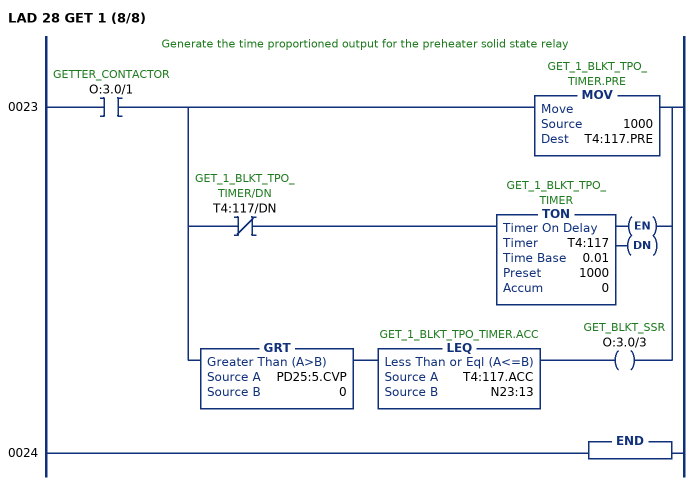
% Rung: 23 %
% Generate the time proportioned output for the preheater solid state relay %
SOR XIC O:3.0/1 BST MOV 1000 T4:117.PRE NXB XIO T4:117/DN TON T4:117 0.01 1000 0 NXB GRT PD25:5.CVP 0 LEQ T4:117.ACC N23:13 OTE O:3.0/3 BND EOR
%   O:3.0/1  GETTER_CONTACTOR %
%   T4:117  GET_1_BLKT_TPO_TIMER %
%   N23:13  GET_1_BLKT_OUTPUT %
%   O:3.0/3  GET_BLKT_SSR %
% Rung: 24 %
SOR END EOR

LADDER 29 "P CONVERT"    % Pressure Unit Conversions %
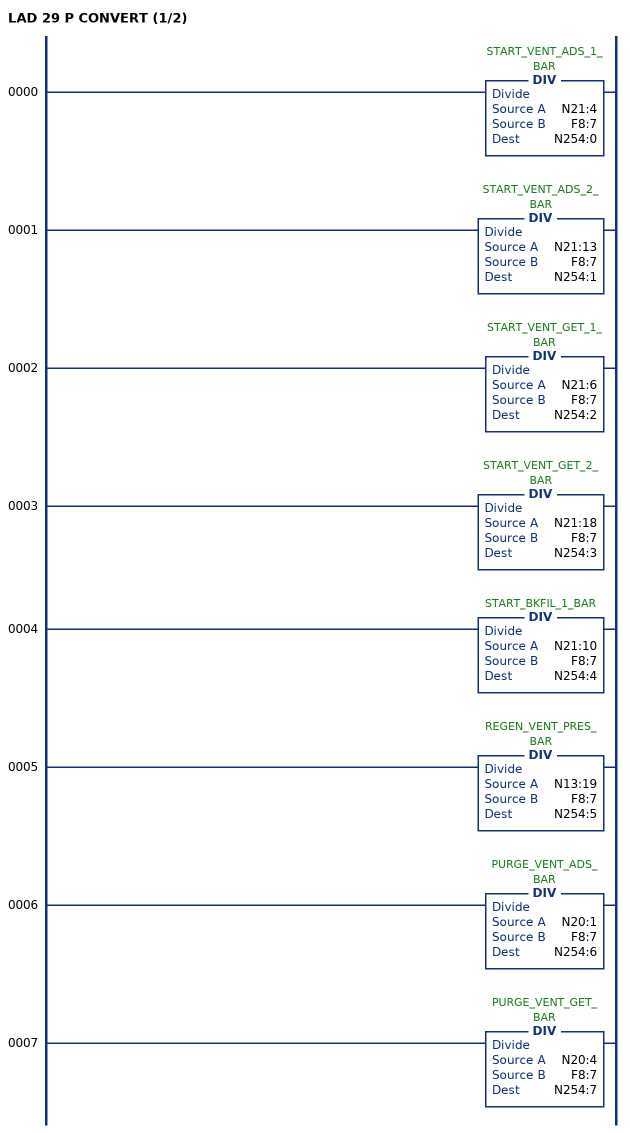
% Rung: 0 %
SOR DIV N21:4 F8:7 N254:0 EOR
%   N21:4  START_VENT_ADS_1_PRS %
%   F8:7  BAR_DIV_FLOAT %
%   N254:0  START_VENT_ADS_1_BAR %
% Rung: 1 %
SOR DIV N21:13 F8:7 N254:1 EOR
%   N21:13  START_VENT_ADS_2_PRS %
%   F8:7  BAR_DIV_FLOAT %
%   N254:1  START_VENT_ADS_2_BAR %
% Rung: 2 %
SOR DIV N21:6 F8:7 N254:2 EOR
%   N21:6  START_VENT_GET_1_PRS %
%   F8:7  BAR_DIV_FLOAT %
%   N254:2  START_VENT_GET_1_BAR %
% Rung: 3 %
SOR DIV N21:18 F8:7 N254:3 EOR
%   N21:18  START_VENT_GET_2_PRS %
%   F8:7  BAR_DIV_FLOAT %
%   N254:3  START_VENT_GET_2_BAR %
% Rung: 4 %
SOR DIV N21:10 F8:7 N254:4 EOR
%   N21:10  START_BKFIL_1_PRS %
%   F8:7  BAR_DIV_FLOAT %
%   N254:4  START_BKFIL_1_BAR %
% Rung: 5 %
SOR DIV N13:19 F8:7 N254:5 EOR
%   N13:19  REGEN_VENT_PRES %
%   F8:7  BAR_DIV_FLOAT %
%   N254:5  REGEN_VENT_PRES_BAR %
% Rung: 6 %
SOR DIV N20:1 F8:7 N254:6 EOR
%   N20:1  PURGE_VENT_ADS_PRES %
%   F8:7  BAR_DIV_FLOAT %
%   N254:6  PURGE_VENT_ADS_BAR %
% Rung: 7 %
SOR DIV N20:4 F8:7 N254:7 EOR
%   N20:4  PURGE_VENT_GET_PRES %
%   F8:7  BAR_DIV_FLOAT %
%   N254:7  PURGE_VENT_GET_BAR %

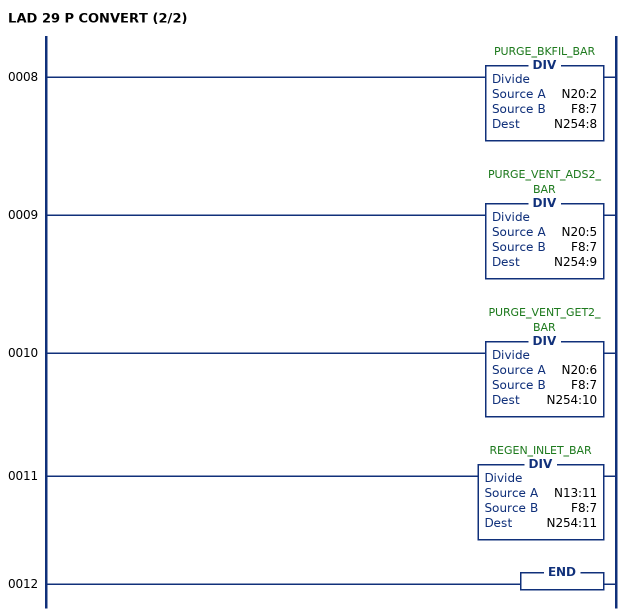
% Rung: 8 %
SOR DIV N20:2 F8:7 N254:8 EOR
%   N20:2  PURGE_BKFIL_PRES %
%   F8:7  BAR_DIV_FLOAT %
%   N254:8  PURGE_BKFIL_BAR %
% Rung: 9 %
SOR DIV N20:5 F8:7 N254:9 EOR
%   N20:5  PURGE_VENT_ADS_2_PX %
%   F8:7  BAR_DIV_FLOAT %
%   N254:9  PURGE_VENT_ADS2_BAR %
% Rung: 10 %
SOR DIV N20:6 F8:7 N254:10 EOR
%   N20:6  PURGE_VENT_GET_2_PX %
%   F8:7  BAR_DIV_FLOAT %
%   N254:10  PURGE_VENT_GET2_BAR %
% Rung: 11 %
SOR DIV N13:11 F8:7 N254:11 EOR
%   N13:11  REGEN_INLET_PSIG %
%   F8:7  BAR_DIV_FLOAT %
%   N254:11  REGEN_INLET_BAR %
% Rung: 12 %
SOR END EOR

LADDER 49 "MODBUS"
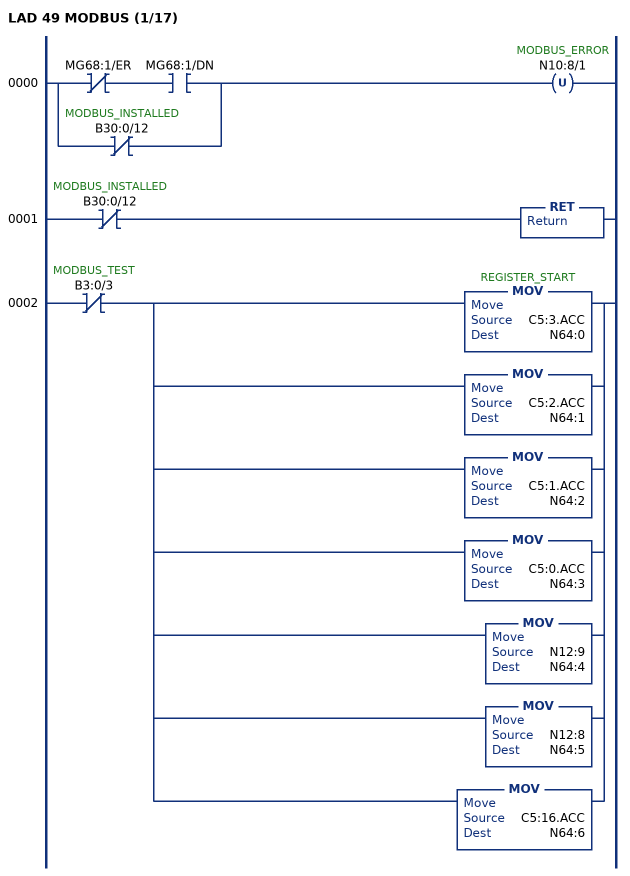
% Rung: 0 %
SOR BST XIO MG68:1/ER XIC MG68:1/DN NXB XIO B30:0/12 BND OTU N10:8/1 EOR
%   B30:0/12  MODBUS_INSTALLED %
%   N10:8/1  MODBUS_ERROR %
% Rung: 1 %
SOR XIO B30:0/12 RET EOR
%   B30:0/12  MODBUS_INSTALLED %
% Rung: 2 %
SOR XIO B3:0/3 BST MOV C5:3.ACC N64:0 NXB MOV C5:2.ACC N64:1 NXB MOV C5:1.ACC N64:2 NXB MOV C5:0.ACC N64:3 NXB MOV N12:9 N64:4 NXB MOV N12:8 N64:5 NXB MOV C5:16.ACC N64:6 BND EOR
%   B3:0/3  MODBUS_TEST %
%   C5:3  PURIFY_ACTIVE_TTL_DY  "COUNTER The number of total elapsed purification days for the process equipment" %
%   N64:0  REGISTER_START %
%   C5:2  PURIFY_ACTIVE_TTL_HR  "COUNTER The number of total elapsed purification hours for the process equipment" %
%   C5:1  PURIFY_ACTIVE_MINUTE  "COUNTER The number of elapsed purification minutes for the current ADS (60 min)" %
%   C5:0  PURIFY_ACTIVE_HOURS  "COUNTER The number of elapsed purification hours for the current ADS" %
%   N12:9  MIN_LEFT_IN_PURIFY %
%   N12:8  HRS_LEFT_IN_PURIFY %
%   C5:16  GETTER_SERVICE_DAYS %

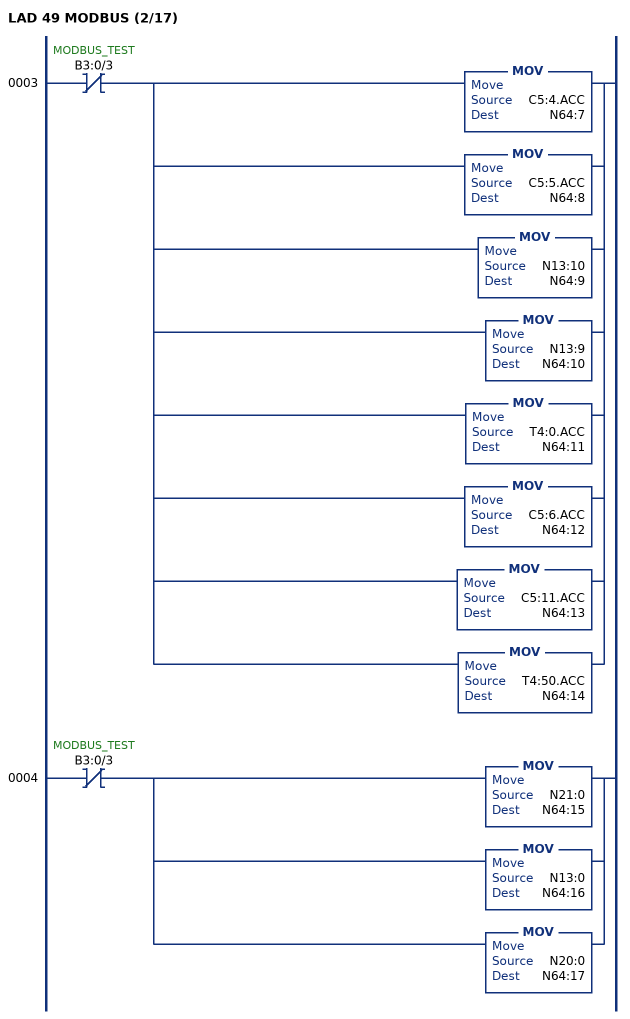
% Rung: 3 %
SOR XIO B3:0/3 BST MOV C5:4.ACC N64:7 NXB MOV C5:5.ACC N64:8 NXB MOV N13:10 N64:9 NXB MOV N13:9 N64:10 NXB MOV T4:0.ACC N64:11 NXB MOV C5:6.ACC N64:12 NXB MOV C5:11.ACC N64:13 NXB MOV T4:50.ACC N64:14 BND EOR
%   B3:0/3  MODBUS_TEST %
%   C5:4  REGEN_RUN_MINUTE %
%   C5:5  REGEN_COOL_MINUTE  "COUNTER Regen the number of minutes for which the bed has cooled" %
%   N13:10  REGEN_MIN_LEFT  "STATUS Preheater Alarm Measured temperature change" %
%   N13:9  REGEN_HRS_LEFT  "STATUS Regen Preheater Temperature Initial Temperature" %
%   T4:0  PURIFY_OVERLAP_TIMER  "TIMER Purify Overlap" %
%   C5:6  START_PURGE_CTR %
%   C5:11  H2_LEAK_RST_MIN %
%   T4:50  H2_LEAK_RST_SEC %
% Rung: 4 %
SOR XIO B3:0/3 BST MOV N21:0 N64:15 NXB MOV N13:0 N64:16 NXB MOV N20:0 N64:17 BND EOR
%   B3:0/3  MODBUS_TEST %
%   N21:0  START_STATE %
%   N13:0  REGEN_STATE  "STATE The current state of the regen process" %
%   N20:0  PURGE_STATE %

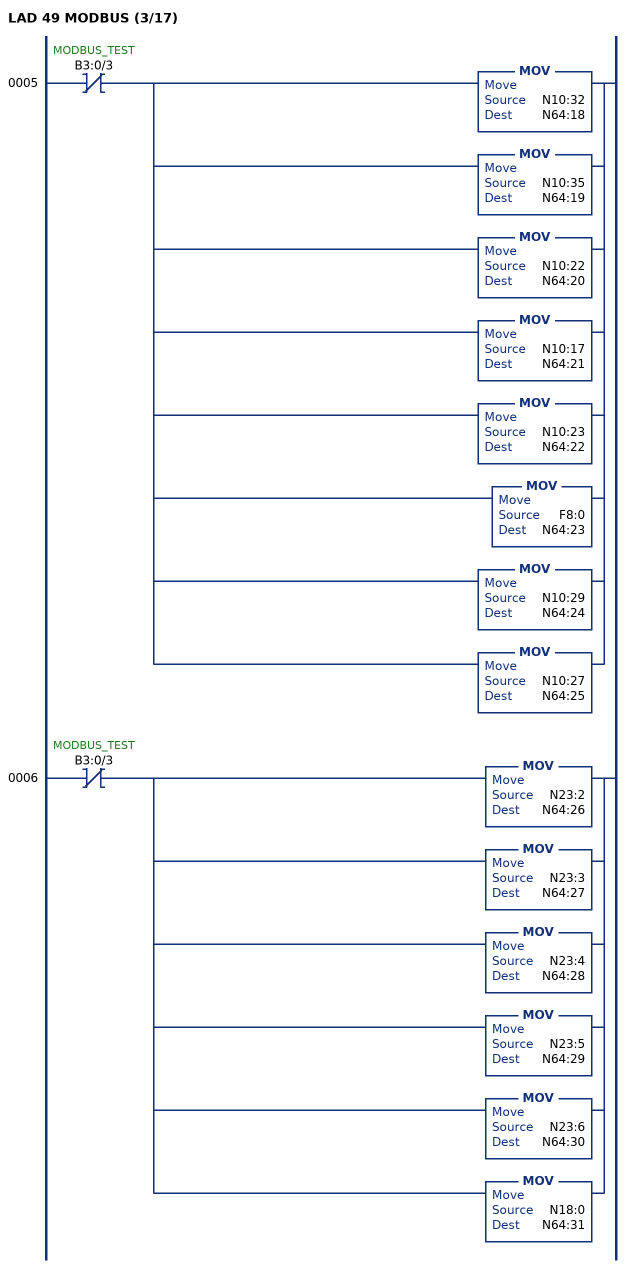
% Rung: 5 %
SOR XIO B3:0/3 BST MOV N10:32 N64:18 NXB MOV N10:35 N64:19 NXB MOV N10:22 N64:20 NXB MOV N10:17 N64:21 NXB MOV N10:23 N64:22 NXB MOV F8:0 N64:23 NXB MOV N10:29 N64:24 NXB MOV N10:27 N64:25 BND EOR
%   B3:0/3  MODBUS_TEST %
%   N10:32  ADS_A_INLET_PX_PRES %
%   N10:35  ADS_B_INLET_PX_PRES %
%   N10:22  OUTLET_PX_PRESSURE %
%   N10:17  INLET_PX_PRESSURE %
%   N10:23  H2_LEVEL_PERCENT %
%   F8:0  MFM_CUM_HR %
%   N10:29  MFC_SLPM %
%   N10:27  MFC_SETPOINT %
% Rung: 6 %
SOR XIO B3:0/3 BST MOV N23:2 N64:26 NXB MOV N23:3 N64:27 NXB MOV N23:4 N64:28 NXB MOV N23:5 N64:29 NXB MOV N23:6 N64:30 NXB MOV N18:0 N64:31 BND EOR
%   B3:0/3  MODBUS_TEST %
%   N23:2  GET_1_PH_INNER_TEMP %
%   N23:3  GET_1_PH_OUTER_TEMP %
%   N23:4  GET_1_PH_GAS_TEMP %
%   N23:5  GET_1_VSL_WALL_TEMP %
%   N23:6  GET_1_VSL_BED_TEMP %
%   N18:0  GET_VSL_OUT_GAS_TEMP %

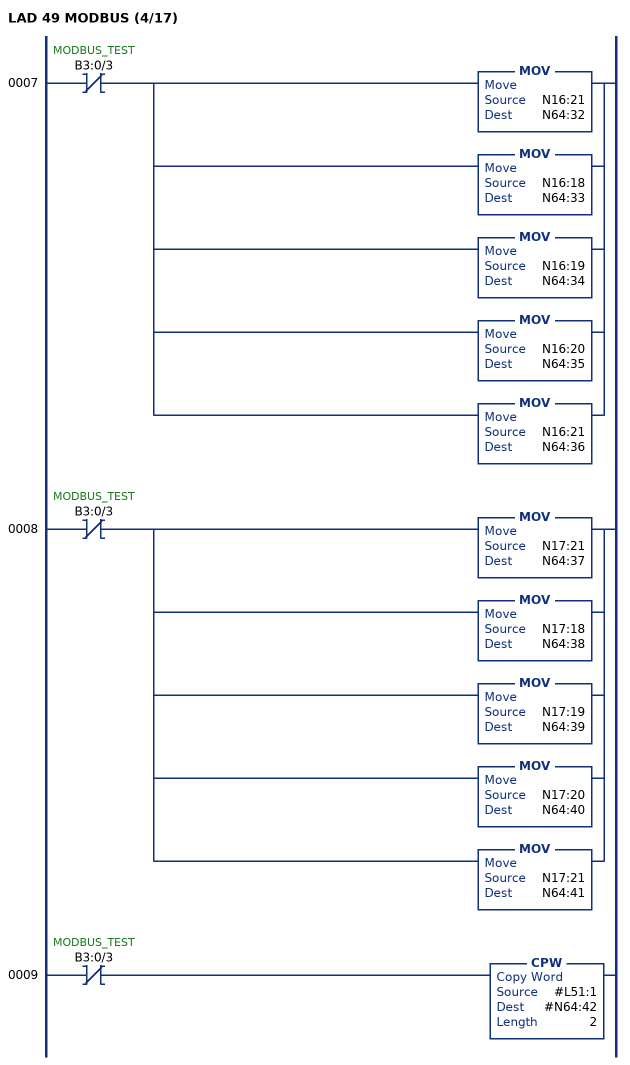
% Rung: 7 %
SOR XIO B3:0/3 BST MOV N16:21 N64:32 NXB MOV N16:18 N64:33 NXB MOV N16:19 N64:34 NXB MOV N16:20 N64:35 NXB MOV N16:21 N64:36 BND EOR
%   B3:0/3  MODBUS_TEST %
%   N16:21  ADS_A_BED_TEMP_READ %
%   N16:18  PH_A_WALL_TEMP_READ %
%   N16:19  PH_A_GAS_TEMP_READ %
%   N16:20  ADS_A_WALL_TEMP_READ %
% Rung: 8 %
SOR XIO B3:0/3 BST MOV N17:21 N64:37 NXB MOV N17:18 N64:38 NXB MOV N17:19 N64:39 NXB MOV N17:20 N64:40 NXB MOV N17:21 N64:41 BND EOR
%   B3:0/3  MODBUS_TEST %
%   N17:21  ADS_B_BED_TEMP_READ %
%   N17:18  PH_B_WALL_TEMP_READ %
%   N17:19  PH_B_GAS_TEMP_READ %
%   N17:20  ADS_B_WALL_TEMP_READ %
% Rung: 9 %
SOR XIO B3:0/3 CPW #L51:1 #N64:42 2 EOR
%   B3:0/3  MODBUS_TEST %
%   L51:1  TOTAL_FLOW_MODBUS %

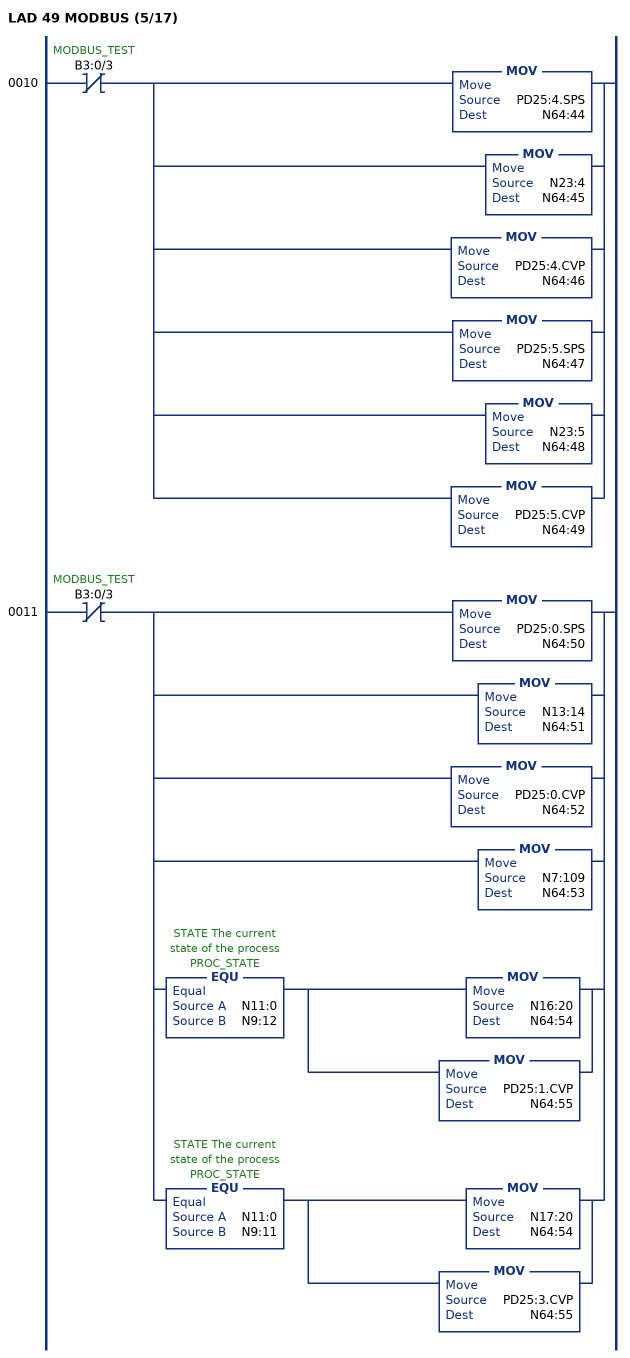
% Rung: 10 %
SOR XIO B3:0/3 BST MOV PD25:4.SPS N64:44 NXB MOV N23:4 N64:45 NXB MOV PD25:4.CVP N64:46 NXB MOV PD25:5.SPS N64:47 NXB MOV N23:5 N64:48 NXB MOV PD25:5.CVP N64:49 BND EOR
%   B3:0/3  MODBUS_TEST %
%   N23:4  GET_1_PH_GAS_TEMP %
%   N23:5  GET_1_VSL_WALL_TEMP %
% Rung: 11 %
SOR XIO B3:0/3 BST MOV PD25:0.SPS N64:50 NXB MOV N13:14 N64:51 NXB MOV PD25:0.CVP N64:52 NXB MOV N7:109 N64:53 NXB EQU N11:0 N9:12 BST MOV N16:20 N64:54 NXB MOV PD25:1.CVP N64:55 BND NXB EQU N11:0 N9:11 BST MOV N17:20 N64:54 NXB MOV PD25:3.CVP N64:55 BND BND EOR
%   B3:0/3  MODBUS_TEST %
%   N13:14  ADS_PH_GAS_TC %
%   N7:109  BLANKET_SP  "CONTROL Blanket PID Setpoint" %
%   N11:0  PROC_STATE  "STATE The current state of the process" %
%   N9:12  PROC_PFY_B_REG_A  "STATE Process Purify B" %
%   N16:20  ADS_A_WALL_TEMP_READ %
%   N9:11  PROC_PFY_A_REG_B  "STATE Process Purify A" %
%   N17:20  ADS_B_WALL_TEMP_READ %

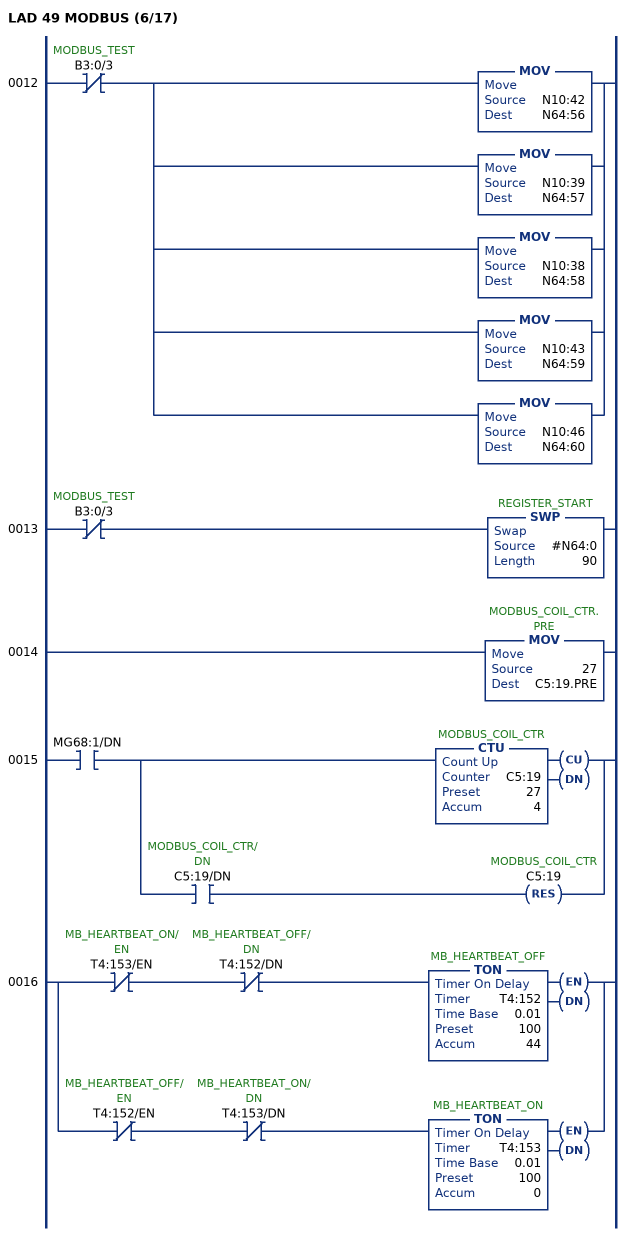
% Rung: 12 %
SOR XIO B3:0/3 BST MOV N10:42 N64:56 NXB MOV N10:39 N64:57 NXB MOV N10:38 N64:58 NXB MOV N10:43 N64:59 NXB MOV N10:46 N64:60 BND EOR
%   B3:0/3  MODBUS_TEST %
%   N10:42  ARGON_PX_PRESS %
%   N10:39  WATER_FLOW_GPM %
%   N10:38  PNEU_PX_PRESS %
%   N10:43  PIPING_BAY_WC %
%   N10:46  ELEC_CAB_WC %
% Rung: 13 %
SOR XIO B3:0/3 SWP #N64:0 90 EOR
%   B3:0/3  MODBUS_TEST %
%   N64:0  REGISTER_START %
% Rung: 14 %
SOR MOV 27 C5:19.PRE EOR
%   C5:19  MODBUS_COIL_CTR %
% Rung: 15 %
SOR XIC MG68:1/DN BST CTU C5:19 27 4 NXB XIC C5:19/DN RES C5:19 BND EOR
%   C5:19  MODBUS_COIL_CTR %
% Rung: 16 %
SOR BST XIO T4:153/EN XIO T4:152/DN TON T4:152 0.01 100 44 NXB XIO T4:152/EN XIO T4:153/DN TON T4:153 0.01 100 0 BND EOR
%   T4:153  MB_HEARTBEAT_ON %
%   T4:152  MB_HEARTBEAT_OFF %

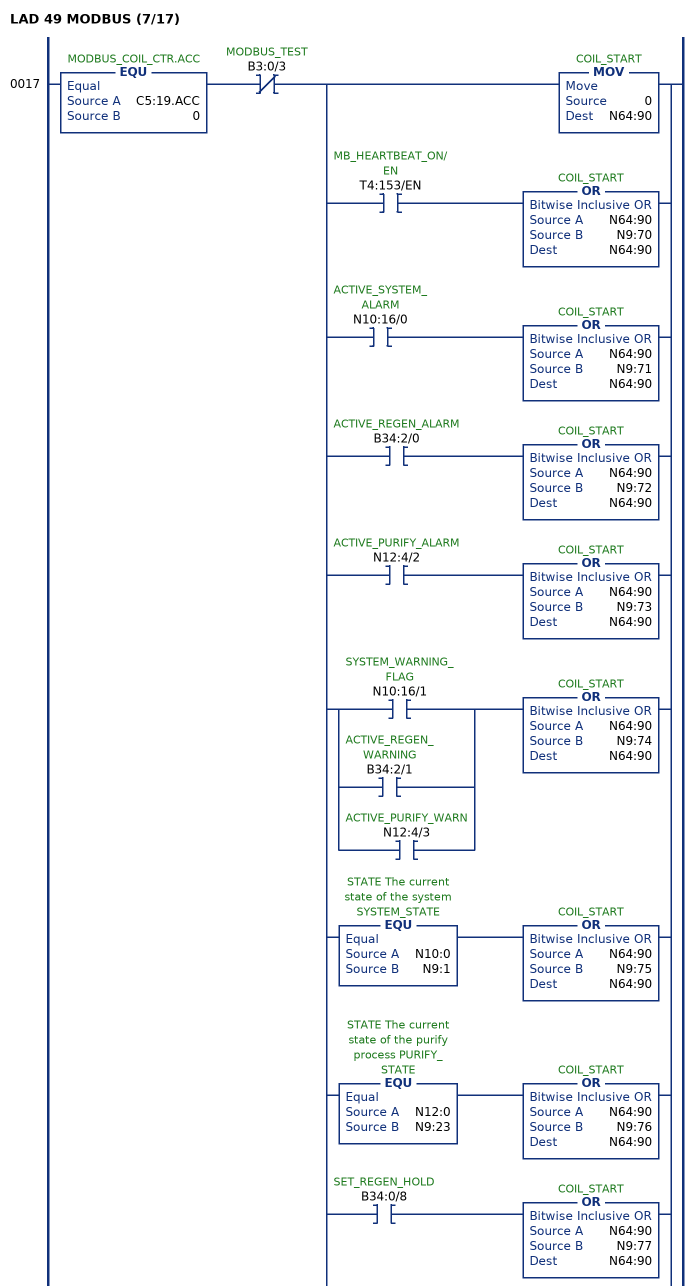

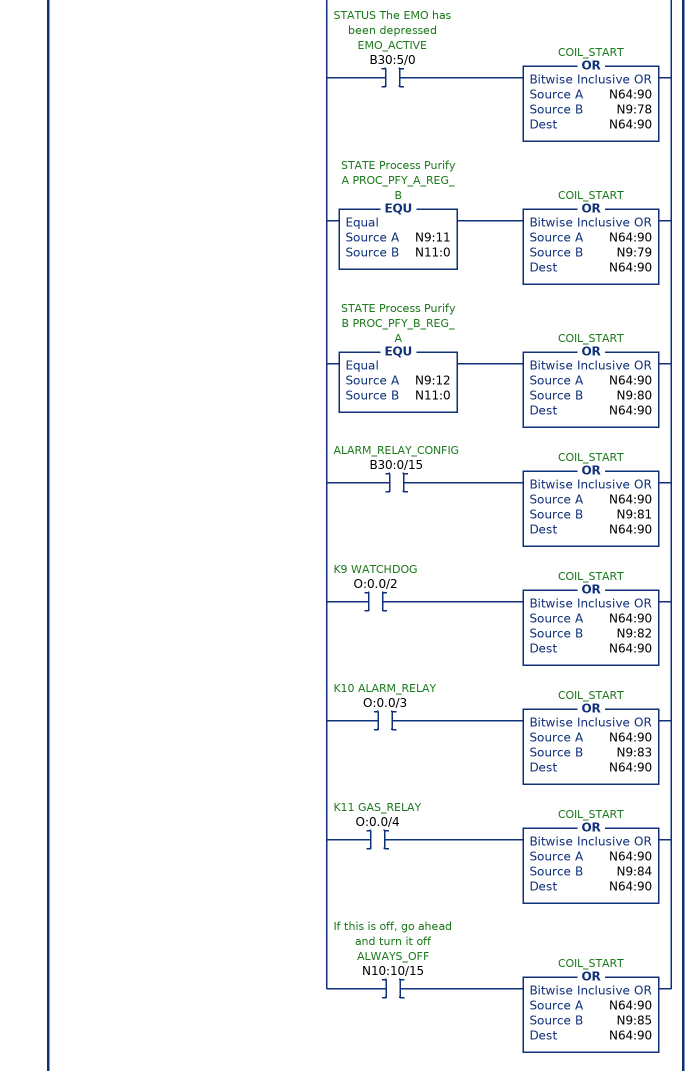
% Rung: 17 %
SOR EQU C5:19.ACC 0 XIO B3:0/3 BST MOV 0 N64:90 NXB XIC T4:153/EN OR N64:90 N9:70 N64:90 NXB XIC N10:16/0 OR N64:90 N9:71 N64:90 NXB XIC B34:2/0 OR N64:90 N9:72 N64:90 NXB XIC N12:4/2 OR N64:90 N9:73 N64:90 NXB BST XIC N10:16/1 NXB XIC B34:2/1 NXB XIC N12:4/3 BND OR N64:90 N9:74 N64:90 NXB EQU N10:0 N9:1 OR N64:90 N9:75 N64:90 NXB EQU N12:0 N9:23 OR N64:90 N9:76 N64:90 NXB XIC B34:0/8 OR N64:90 N9:77 N64:90 NXB XIC B30:5/0 OR N64:90 N9:78 N64:90 NXB EQU N9:11 N11:0 OR N64:90 N9:79 N64:90 NXB EQU N9:12 N11:0 OR N64:90 N9:80 N64:90 NXB XIC B30:0/15 OR N64:90 N9:81 N64:90 NXB XIC O:0.0/2 OR N64:90 N9:82 N64:90 NXB XIC O:0.0/3 OR N64:90 N9:83 N64:90 NXB XIC O:0.0/4 OR N64:90 N9:84 N64:90 NXB XIC N10:10/15 OR N64:90 N9:85 N64:90 BND EOR
%   C5:19  MODBUS_COIL_CTR %
%   B3:0/3  MODBUS_TEST %
%   N64:90  COIL_START %
%   T4:153  MB_HEARTBEAT_ON %
%   N9:70  BIT_0 %
%   N10:16/0  ACTIVE_SYSTEM_ALARM %
%   N9:71  BIT_1 %
%   B34:2/0  ACTIVE_REGEN_ALARM %
%   N9:72  BIT_2 %
%   N12:4/2  ACTIVE_PURIFY_ALARM %
%   N9:73  BIT_3 %
%   N10:16/1  SYSTEM_WARNING_FLAG %
%   B34:2/1  ACTIVE_REGEN_WARNING %
%   N12:4/3  ACTIVE_PURIFY_WARN %
%   N9:74  BIT_4 %
%   N10:0  SYSTEM_STATE  "STATE The current state of the system" %
%   N9:1  SYSTEM_STANDBY  "STATE System Process" %
%   N9:75  BIT_5 %
%   N12:0  PURIFY_STATE  "STATE The current state of the purify process" %
%   N9:23  PURIFY_MANUAL_HOLD  "STATE Purify Manual Hold" %
%   N9:76  BIT_6 %
%   B34:0/8  SET_REGEN_HOLD %
%   N9:77  BIT_7 %
%   B30:5/0  EMO_ACTIVE  "STATUS The EMO has been depressed" %
%   N9:78  BIT_8 %
%   N9:11  PROC_PFY_A_REG_B  "STATE Process Purify A" %
%   N11:0  PROC_STATE  "STATE The current state of the process" %
%   N9:79  BIT_9 %
%   N9:12  PROC_PFY_B_REG_A  "STATE Process Purify B" %
%   N9:80  BIT_10 %
%   B30:0/15  ALARM_RELAY_CONFIG %
%   N9:81  BIT_11 %
%   O:0.0/2  WATCHDOG  "K9" %
%   N9:82  BIT_12 %
%   O:0.0/3  ALARM_RELAY  "K10" %
%   N9:83  BIT_13 %
%   O:0.0/4  GAS_RELAY  "K11" %
%   N9:84  BIT_14 %
%   N10:10/15  ALWAYS_OFF  "If this is off, go ahead and turn it off" %
%   N9:85  BIT_15 %

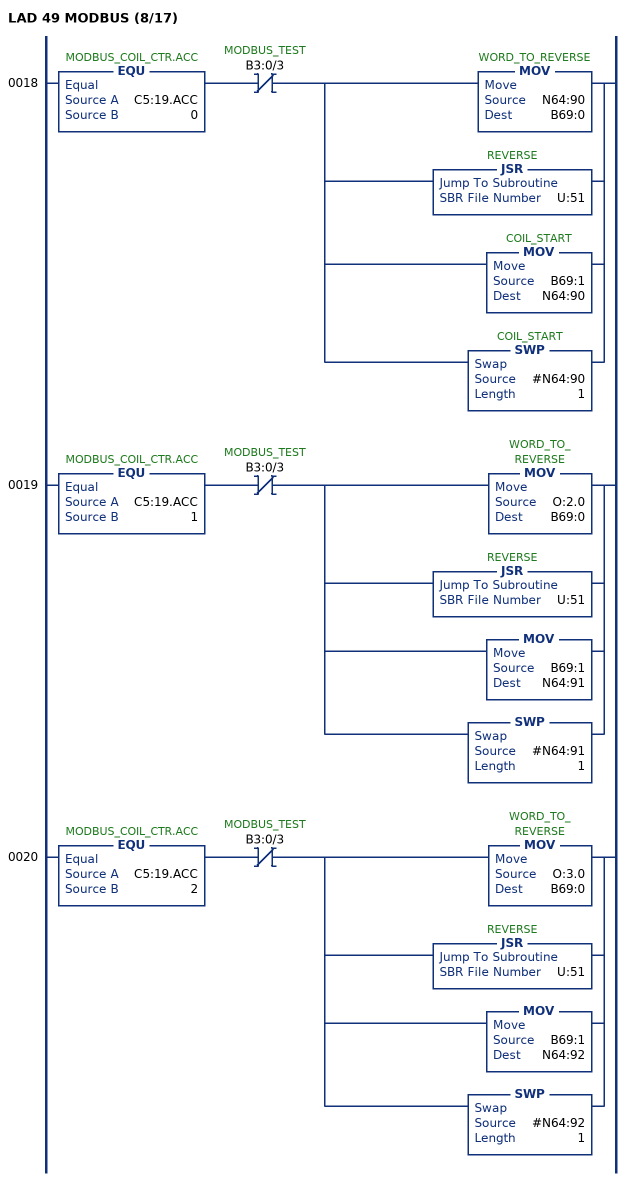
% Rung: 18 %
SOR EQU C5:19.ACC 0 XIO B3:0/3 BST MOV N64:90 B69:0 NXB JSR U:51 NXB MOV B69:1 N64:90 NXB SWP #N64:90 1 BND EOR
%   C5:19  MODBUS_COIL_CTR %
%   B3:0/3  MODBUS_TEST %
%   N64:90  COIL_START %
%   B69:0  WORD_TO_REVERSE %
%   U:51  REVERSE %
%   B69:1  REVERSED_WORD %
% Rung: 19 %
SOR EQU C5:19.ACC 1 XIO B3:0/3 BST MOV O:2.0 B69:0 NXB JSR U:51 NXB MOV B69:1 N64:91 NXB SWP #N64:91 1 BND EOR
%   C5:19  MODBUS_COIL_CTR %
%   B3:0/3  MODBUS_TEST %
%   B69:0  WORD_TO_REVERSE %
%   U:51  REVERSE %
%   B69:1  REVERSED_WORD %
% Rung: 20 %
SOR EQU C5:19.ACC 2 XIO B3:0/3 BST MOV O:3.0 B69:0 NXB JSR U:51 NXB MOV B69:1 N64:92 NXB SWP #N64:92 1 BND EOR
%   C5:19  MODBUS_COIL_CTR %
%   B3:0/3  MODBUS_TEST %
%   B69:0  WORD_TO_REVERSE %
%   U:51  REVERSE %
%   B69:1  REVERSED_WORD %

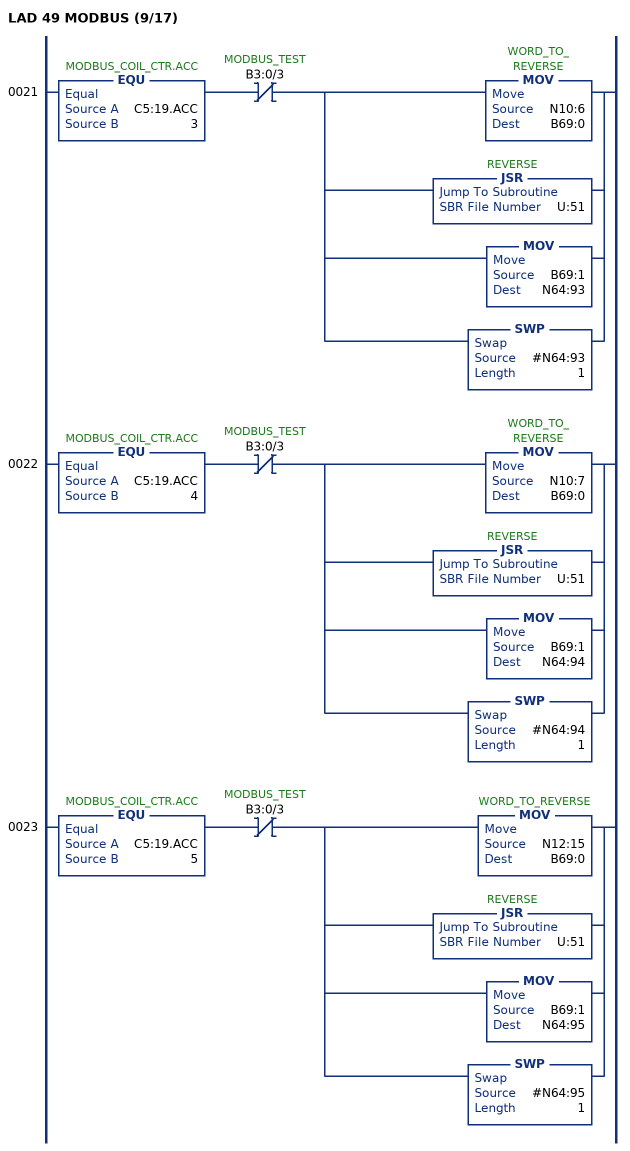
% Rung: 21 %
SOR EQU C5:19.ACC 3 XIO B3:0/3 BST MOV N10:6 B69:0 NXB JSR U:51 NXB MOV B69:1 N64:93 NXB SWP #N64:93 1 BND EOR
%   C5:19  MODBUS_COIL_CTR %
%   B3:0/3  MODBUS_TEST %
%   N10:6  SYSTEM_ALARMS_0  "ALARM System alarms" %
%   B69:0  WORD_TO_REVERSE %
%   U:51  REVERSE %
%   B69:1  REVERSED_WORD %
% Rung: 22 %
SOR EQU C5:19.ACC 4 XIO B3:0/3 BST MOV N10:7 B69:0 NXB JSR U:51 NXB MOV B69:1 N64:94 NXB SWP #N64:94 1 BND EOR
%   C5:19  MODBUS_COIL_CTR %
%   B3:0/3  MODBUS_TEST %
%   N10:7  SYSTEM_ALARMS_1  "ALARM System alarms" %
%   B69:0  WORD_TO_REVERSE %
%   U:51  REVERSE %
%   B69:1  REVERSED_WORD %
% Rung: 23 %
SOR EQU C5:19.ACC 5 XIO B3:0/3 BST MOV N12:15 B69:0 NXB JSR U:51 NXB MOV B69:1 N64:95 NXB SWP #N64:95 1 BND EOR
%   C5:19  MODBUS_COIL_CTR %
%   B3:0/3  MODBUS_TEST %
%   N12:15  PURIFY_ALARMS_0 %
%   B69:0  WORD_TO_REVERSE %
%   U:51  REVERSE %
%   B69:1  REVERSED_WORD %

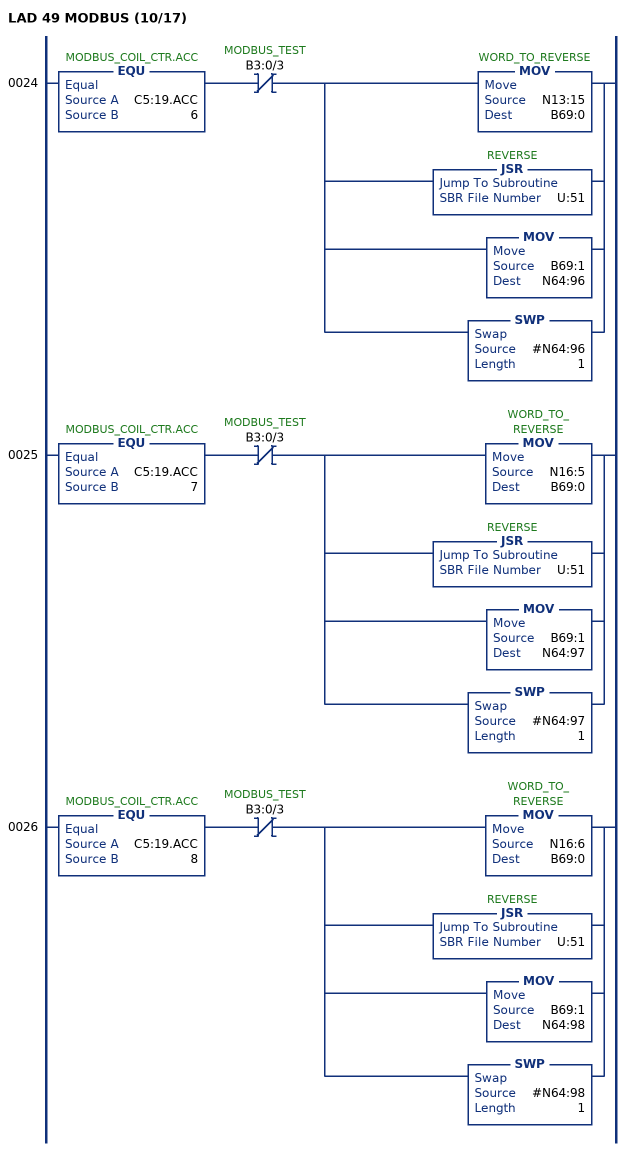
% Rung: 24 %
SOR EQU C5:19.ACC 6 XIO B3:0/3 BST MOV N13:15 B69:0 NXB JSR U:51 NXB MOV B69:1 N64:96 NXB SWP #N64:96 1 BND EOR
%   C5:19  MODBUS_COIL_CTR %
%   B3:0/3  MODBUS_TEST %
%   N13:15  REGEN_ALARMS_0 %
%   B69:0  WORD_TO_REVERSE %
%   U:51  REVERSE %
%   B69:1  REVERSED_WORD %
% Rung: 25 %
SOR EQU C5:19.ACC 7 XIO B3:0/3 BST MOV N16:5 B69:0 NXB JSR U:51 NXB MOV B69:1 N64:97 NXB SWP #N64:97 1 BND EOR
%   C5:19  MODBUS_COIL_CTR %
%   B3:0/3  MODBUS_TEST %
%   N16:5  ADS_A_REGEN_ALARMS_0  "ALARM ADS A Alarms" %
%   B69:0  WORD_TO_REVERSE %
%   U:51  REVERSE %
%   B69:1  REVERSED_WORD %
% Rung: 26 %
SOR EQU C5:19.ACC 8 XIO B3:0/3 BST MOV N16:6 B69:0 NXB JSR U:51 NXB MOV B69:1 N64:98 NXB SWP #N64:98 1 BND EOR
%   C5:19  MODBUS_COIL_CTR %
%   B3:0/3  MODBUS_TEST %
%   N16:6  ADS_A_PURIFY_ALARMS  "ALARM ADS A Alarms" %
%   B69:0  WORD_TO_REVERSE %
%   U:51  REVERSE %
%   B69:1  REVERSED_WORD %

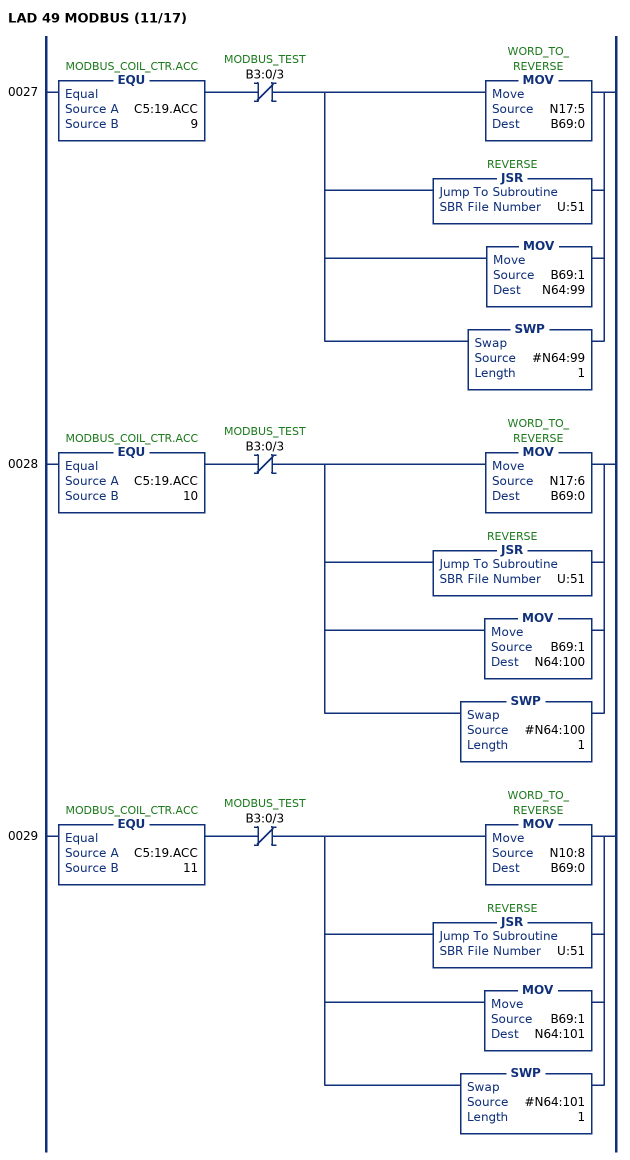
% Rung: 27 %
SOR EQU C5:19.ACC 9 XIO B3:0/3 BST MOV N17:5 B69:0 NXB JSR U:51 NXB MOV B69:1 N64:99 NXB SWP #N64:99 1 BND EOR
%   C5:19  MODBUS_COIL_CTR %
%   B3:0/3  MODBUS_TEST %
%   N17:5  ADS_B_REGEN_ALARMS_0  "ALARM Alarm bits" %
%   B69:0  WORD_TO_REVERSE %
%   U:51  REVERSE %
%   B69:1  REVERSED_WORD %
% Rung: 28 %
SOR EQU C5:19.ACC 10 XIO B3:0/3 BST MOV N17:6 B69:0 NXB JSR U:51 NXB MOV B69:1 N64:100 NXB SWP #N64:100 1 BND EOR
%   C5:19  MODBUS_COIL_CTR %
%   B3:0/3  MODBUS_TEST %
%   N17:6  ADS_B_PURIFY_ALARMS  "ALARM ADS B Alarms" %
%   B69:0  WORD_TO_REVERSE %
%   U:51  REVERSE %
%   B69:1  REVERSED_WORD %
% Rung: 29 %
SOR EQU C5:19.ACC 11 XIO B3:0/3 BST MOV N10:8 B69:0 NXB JSR U:51 NXB MOV B69:1 N64:101 NXB SWP #N64:101 1 BND EOR
%   C5:19  MODBUS_COIL_CTR %
%   B3:0/3  MODBUS_TEST %
%   N10:8  SYSTEM_WARNINGS_0  "WARNING System Warnings" %
%   B69:0  WORD_TO_REVERSE %
%   U:51  REVERSE %
%   B69:1  REVERSED_WORD %

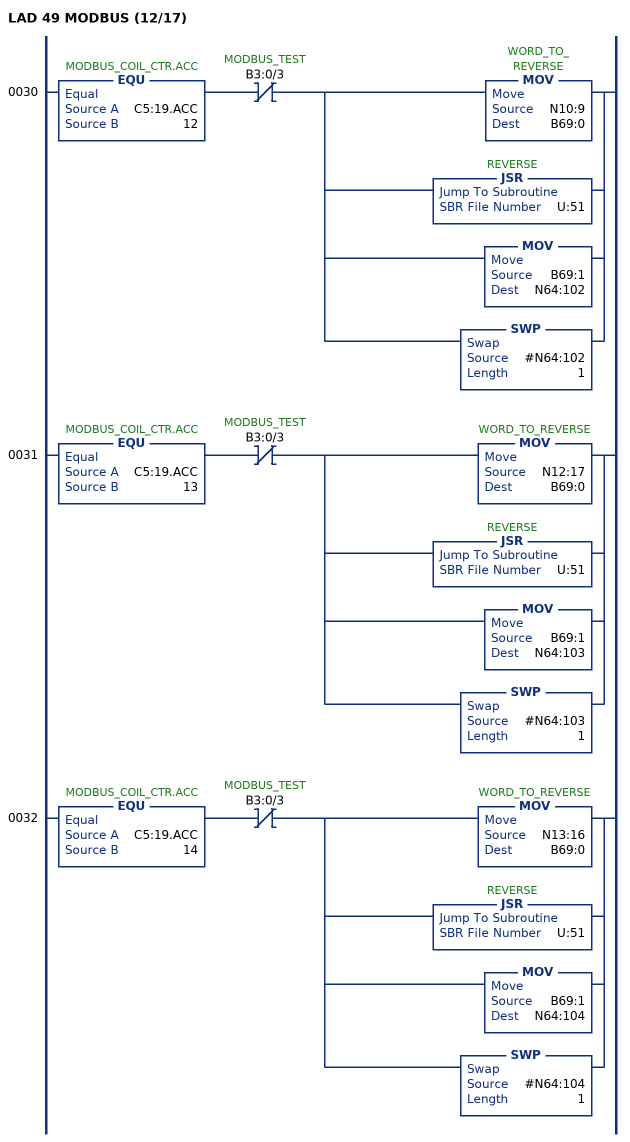
% Rung: 30 %
SOR EQU C5:19.ACC 12 XIO B3:0/3 BST MOV N10:9 B69:0 NXB JSR U:51 NXB MOV B69:1 N64:102 NXB SWP #N64:102 1 BND EOR
%   C5:19  MODBUS_COIL_CTR %
%   B3:0/3  MODBUS_TEST %
%   N10:9  SYSTEM_WARNINGS_1  "WARNING System Warnings" %
%   B69:0  WORD_TO_REVERSE %
%   U:51  REVERSE %
%   B69:1  REVERSED_WORD %
% Rung: 31 %
SOR EQU C5:19.ACC 13 XIO B3:0/3 BST MOV N12:17 B69:0 NXB JSR U:51 NXB MOV B69:1 N64:103 NXB SWP #N64:103 1 BND EOR
%   C5:19  MODBUS_COIL_CTR %
%   B3:0/3  MODBUS_TEST %
%   N12:17  PURIFY_WARNINGS_0 %
%   B69:0  WORD_TO_REVERSE %
%   U:51  REVERSE %
%   B69:1  REVERSED_WORD %
% Rung: 32 %
SOR EQU C5:19.ACC 14 XIO B3:0/3 BST MOV N13:16 B69:0 NXB JSR U:51 NXB MOV B69:1 N64:104 NXB SWP #N64:104 1 BND EOR
%   C5:19  MODBUS_COIL_CTR %
%   B3:0/3  MODBUS_TEST %
%   N13:16  REGEN_WARNINGS_0 %
%   B69:0  WORD_TO_REVERSE %
%   U:51  REVERSE %
%   B69:1  REVERSED_WORD %

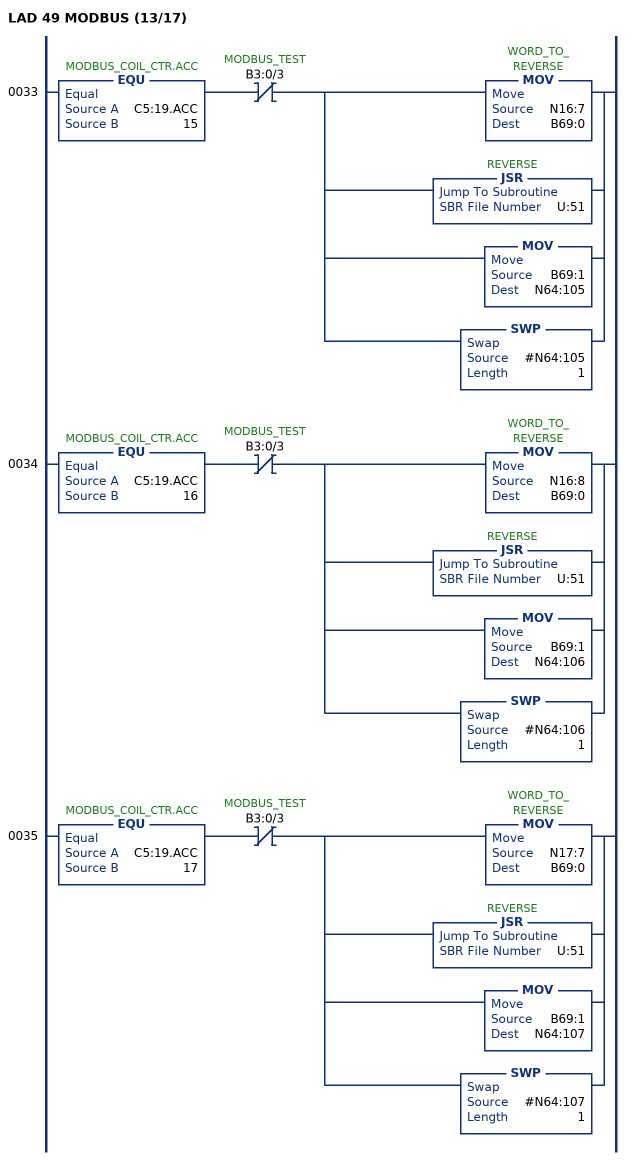
% Rung: 33 %
SOR EQU C5:19.ACC 15 XIO B3:0/3 BST MOV N16:7 B69:0 NXB JSR U:51 NXB MOV B69:1 N64:105 NXB SWP #N64:105 1 BND EOR
%   C5:19  MODBUS_COIL_CTR %
%   B3:0/3  MODBUS_TEST %
%   N16:7  ADS_A_REGEN_WARN_0  "WARNING ADS A Warnings" %
%   B69:0  WORD_TO_REVERSE %
%   U:51  REVERSE %
%   B69:1  REVERSED_WORD %
% Rung: 34 %
SOR EQU C5:19.ACC 16 XIO B3:0/3 BST MOV N16:8 B69:0 NXB JSR U:51 NXB MOV B69:1 N64:106 NXB SWP #N64:106 1 BND EOR
%   C5:19  MODBUS_COIL_CTR %
%   B3:0/3  MODBUS_TEST %
%   N16:8  ADS_A_PURIFY_WARNS  "WARNING ADS A Warnings" %
%   B69:0  WORD_TO_REVERSE %
%   U:51  REVERSE %
%   B69:1  REVERSED_WORD %
% Rung: 35 %
SOR EQU C5:19.ACC 17 XIO B3:0/3 BST MOV N17:7 B69:0 NXB JSR U:51 NXB MOV B69:1 N64:107 NXB SWP #N64:107 1 BND EOR
%   C5:19  MODBUS_COIL_CTR %
%   B3:0/3  MODBUS_TEST %
%   N17:7  ADS_B_REGEN_WARN_0  "WARNING Warning bits" %
%   B69:0  WORD_TO_REVERSE %
%   U:51  REVERSE %
%   B69:1  REVERSED_WORD %

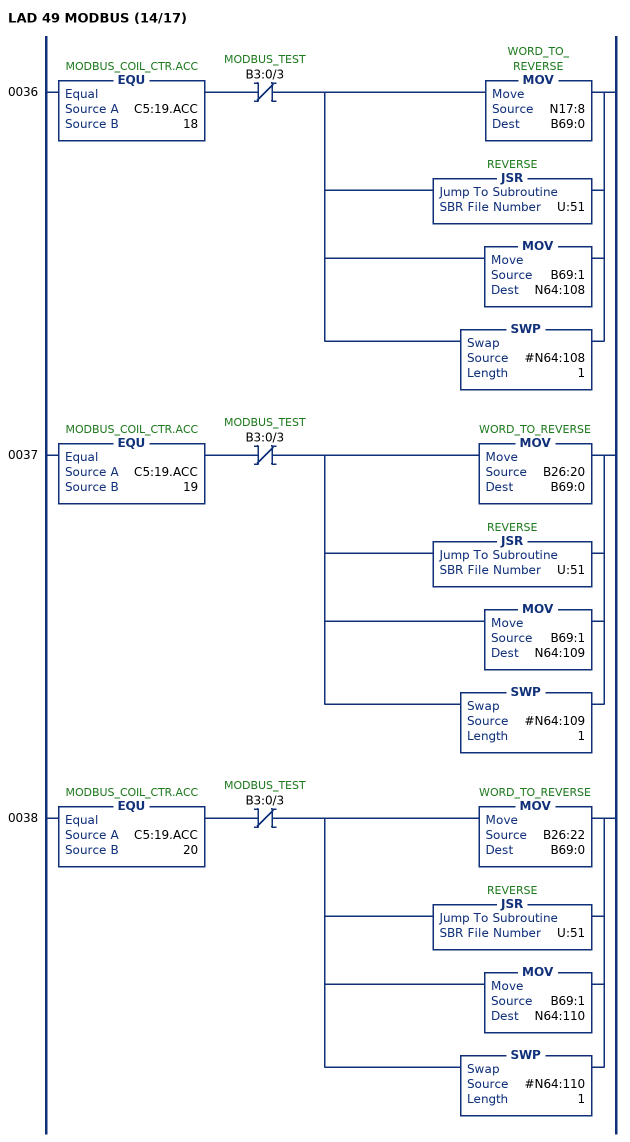
% Rung: 36 %
SOR EQU C5:19.ACC 18 XIO B3:0/3 BST MOV N17:8 B69:0 NXB JSR U:51 NXB MOV B69:1 N64:108 NXB SWP #N64:108 1 BND EOR
%   C5:19  MODBUS_COIL_CTR %
%   B3:0/3  MODBUS_TEST %
%   N17:8  ADS_B_PURIFY_WARNS  "WARNING ADS B Warnings" %
%   B69:0  WORD_TO_REVERSE %
%   U:51  REVERSE %
%   B69:1  REVERSED_WORD %
% Rung: 37 %
SOR EQU C5:19.ACC 19 XIO B3:0/3 BST MOV B26:20 B69:0 NXB JSR U:51 NXB MOV B69:1 N64:109 NXB SWP #N64:109 1 BND EOR
%   C5:19  MODBUS_COIL_CTR %
%   B3:0/3  MODBUS_TEST %
%   B26:20  GETTER_ALARMS %
%   B69:0  WORD_TO_REVERSE %
%   U:51  REVERSE %
%   B69:1  REVERSED_WORD %
% Rung: 38 %
SOR EQU C5:19.ACC 20 XIO B3:0/3 BST MOV B26:22 B69:0 NXB JSR U:51 NXB MOV B69:1 N64:110 NXB SWP #N64:110 1 BND EOR
%   C5:19  MODBUS_COIL_CTR %
%   B3:0/3  MODBUS_TEST %
%   B26:22  GET_1_OPEN_TC_ALARMS %
%   B69:0  WORD_TO_REVERSE %
%   U:51  REVERSE %
%   B69:1  REVERSED_WORD %

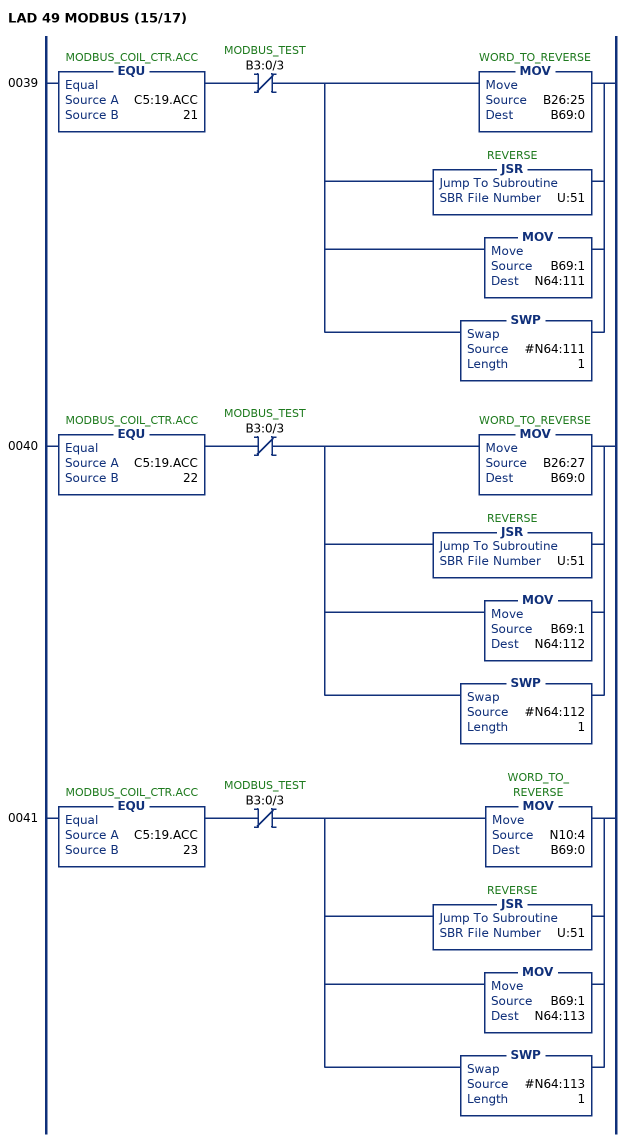
% Rung: 39 %
SOR EQU C5:19.ACC 21 XIO B3:0/3 BST MOV B26:25 B69:0 NXB JSR U:51 NXB MOV B69:1 N64:111 NXB SWP #N64:111 1 BND EOR
%   C5:19  MODBUS_COIL_CTR %
%   B3:0/3  MODBUS_TEST %
%   B26:25  GETTER_WARNINGS %
%   B69:0  WORD_TO_REVERSE %
%   U:51  REVERSE %
%   B69:1  REVERSED_WORD %
% Rung: 40 %
SOR EQU C5:19.ACC 22 XIO B3:0/3 BST MOV B26:27 B69:0 NXB JSR U:51 NXB MOV B69:1 N64:112 NXB SWP #N64:112 1 BND EOR
%   C5:19  MODBUS_COIL_CTR %
%   B3:0/3  MODBUS_TEST %
%   B26:27  GET_1_OPEN_TC_WARNS %
%   B69:0  WORD_TO_REVERSE %
%   U:51  REVERSE %
%   B69:1  REVERSED_WORD %
% Rung: 41 %
SOR EQU C5:19.ACC 23 XIO B3:0/3 BST MOV N10:4 B69:0 NXB JSR U:51 NXB MOV B69:1 N64:113 NXB SWP #N64:113 1 BND EOR
%   C5:19  MODBUS_COIL_CTR %
%   B3:0/3  MODBUS_TEST %
%   N10:4  H2_ALARMS %
%   B69:0  WORD_TO_REVERSE %
%   U:51  REVERSE %
%   B69:1  REVERSED_WORD %

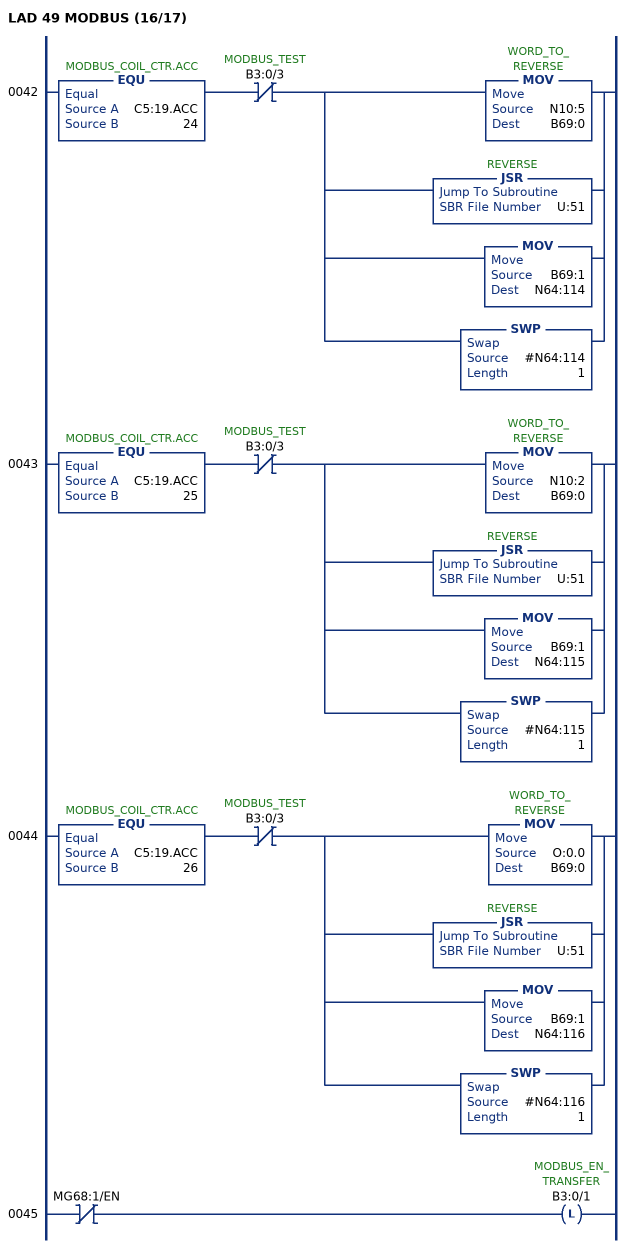
% Rung: 42 %
SOR EQU C5:19.ACC 24 XIO B3:0/3 BST MOV N10:5 B69:0 NXB JSR U:51 NXB MOV B69:1 N64:114 NXB SWP #N64:114 1 BND EOR
%   C5:19  MODBUS_COIL_CTR %
%   B3:0/3  MODBUS_TEST %
%   N10:5  H2_WARNINGS %
%   B69:0  WORD_TO_REVERSE %
%   U:51  REVERSE %
%   B69:1  REVERSED_WORD %
% Rung: 43 %
SOR EQU C5:19.ACC 25 XIO B3:0/3 BST MOV N10:2 B69:0 NXB JSR U:51 NXB MOV B69:1 N64:115 NXB SWP #N64:115 1 BND EOR
%   C5:19  MODBUS_COIL_CTR %
%   B3:0/3  MODBUS_TEST %
%   N10:2  "(LT GETTER SHUTDOWN)" %
%   B69:0  WORD_TO_REVERSE %
%   U:51  REVERSE %
%   B69:1  REVERSED_WORD %
% Rung: 44 %
SOR EQU C5:19.ACC 26 XIO B3:0/3 BST MOV O:0.0 B69:0 NXB JSR U:51 NXB MOV B69:1 N64:116 NXB SWP #N64:116 1 BND EOR
%   C5:19  MODBUS_COIL_CTR %
%   B3:0/3  MODBUS_TEST %
%   B69:0  WORD_TO_REVERSE %
%   U:51  REVERSE %
%   B69:1  REVERSED_WORD %
% Rung: 45 %
SOR XIO MG68:1/EN OTL B3:0/1 EOR
%   B3:0/1  MODBUS_EN_TRANSFER %

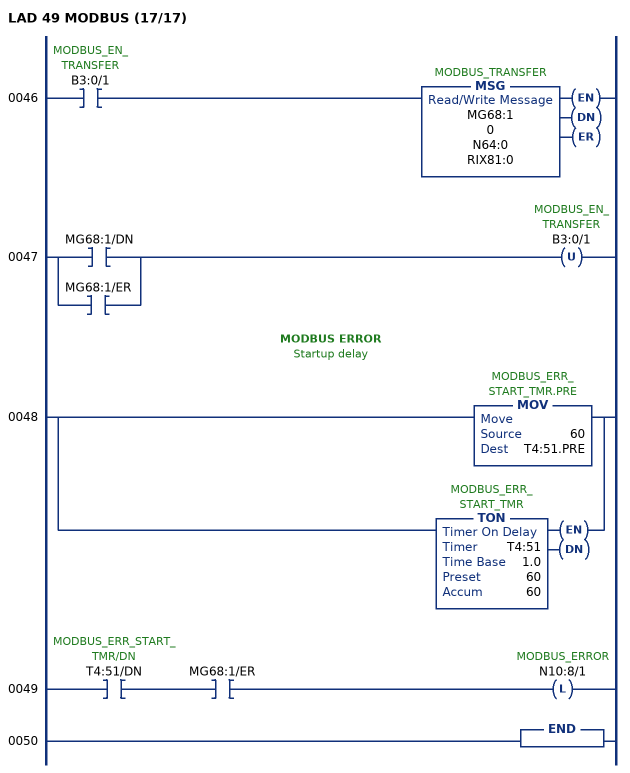
% Rung: 46 %
SOR XIC B3:0/1 MSG MG68:1 0 N64:0 RIX81:0 EOR
%   B3:0/1  MODBUS_EN_TRANSFER %
%   MSG set-up: CIP Generic | 33 | 0 | ? | 0 | 0 | 0 | 0 | 172.16.14.73 | 0 | 0 | 172.16.14.73 | RIX81:0 | 10 | 4 | 150 | 3 | 4 | 96 | 3 | 252 | N64:0 %
%   MG68:1  MODBUS_TRANSFER %
%   N64:0  REGISTER_START %
% Rung: 47 %
SOR BST XIC MG68:1/DN NXB XIC MG68:1/ER BND OTU B3:0/1 EOR
%   B3:0/1  MODBUS_EN_TRANSFER %
% Rung: 48 %
% TITLE: MODBUS ERROR %
% Startup delay %
SOR BST MOV 60 T4:51.PRE NXB TON T4:51 1.0 60 60 BND EOR
%   T4:51  MODBUS_ERR_START_TMR %
% Rung: 49 %
SOR XIC T4:51/DN XIC MG68:1/ER OTL N10:8/1 EOR
%   T4:51  MODBUS_ERR_START_TMR %
%   N10:8/1  MODBUS_ERROR %
% Rung: 50 %
SOR END EOR

LADDER 50 "PLC FAULT"
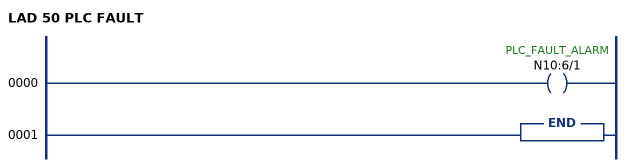
% Rung: 0 %
SOR OTE N10:6/1 EOR
%   N10:6/1  PLC_FAULT_ALARM %
% Rung: 1 %
SOR END EOR

LADDER 51 "REVERSE"
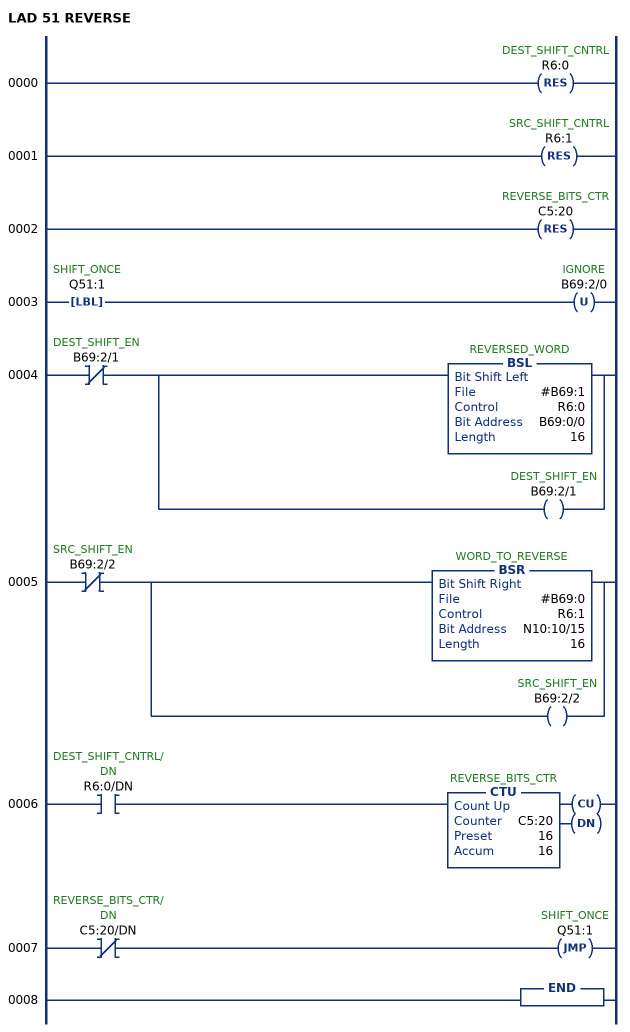
% Rung: 0 %
SOR RES R6:0 EOR
%   R6:0  DEST_SHIFT_CNTRL %
% Rung: 1 %
SOR RES R6:1 EOR
%   R6:1  SRC_SHIFT_CNTRL %
% Rung: 2 %
SOR RES C5:20 EOR
%   C5:20  REVERSE_BITS_CTR %
% Rung: 3 %
SOR LBL Q51:1 OTU B69:2/0 EOR
%   Q51:1  SHIFT_ONCE %
%   B69:2/0  IGNORE %
% Rung: 4 %
SOR XIO B69:2/1 BST BSL #B69:1 R6:0 B69:0/0 16 NXB OTE B69:2/1 BND EOR
%   B69:2/1  DEST_SHIFT_EN %
%   B69:1  REVERSED_WORD %
%   R6:0  DEST_SHIFT_CNTRL %
% Rung: 5 %
SOR XIO B69:2/2 BST BSR #B69:0 R6:1 N10:10/15 16 NXB OTE B69:2/2 BND EOR
%   B69:2/2  SRC_SHIFT_EN %
%   B69:0  WORD_TO_REVERSE %
%   R6:1  SRC_SHIFT_CNTRL %
%   N10:10/15  ALWAYS_OFF  "If this is off, go ahead and turn it off" %
% Rung: 6 %
SOR XIC R6:0/DN CTU C5:20 16 16 EOR
%   R6:0  DEST_SHIFT_CNTRL %
%   C5:20  REVERSE_BITS_CTR %
% Rung: 7 %
SOR XIO C5:20/DN JMP Q51:1 EOR
%   C5:20  REVERSE_BITS_CTR %
%   Q51:1  SHIFT_ONCE %
% Rung: 8 %
SOR END EOR

OTHER DOCUMENTED ADDRESSES
  B3:0/0  TEST
  B3:0/4  PRESSURE_IN_MPA
  B3:0/5  PRESSURE_IN_PSI
  B22:0/0  START_VENT_ADS_1_DN
  B22:0/1  START_VENT_GET_1_DN
  B22:0/2  START_HEAT_GET_DN
  B22:0/3  START_VENT_ALL_DN
  B22:0/4  START_BKFIL_1_DN
  B22:0/5  START_VENT_ADS_2_DN
  B22:0/6  START_VENT_GET_2_DN
  B22:0/7  START_BKFL_2_DN
  B26:0/1  UPS_FAIL_ALM_EN
  B26:1/5  LP_INLET_GAS_ALM_EN
  B26:3  OPEN_TC_ALARM_EN
  B26:3/10  OPEN_TC11_ALARM_EN
  B26:3/15  OPEN_TC16_ALARM_EN
  B26:5/1  UPS_FAIL_WRN_EN
  B26:6/5  LP_INLET_GAS_WRN_EN
  B26:8/11  OPEN_TC11_WARN_EN
  B26:9/0  OPEN_TC16_WARN_EN
  B26:21/0  GET_2_HT_PH_GAS_ALM
  B26:21/1  GET_2_HT_PH_ALARM
  B26:21/2  GET_2_HT_BED_ALARM
  B26:21/3  GET_2_HT_WALL_ALARM
  B26:21/5  GET_2_HTI_ALARM
  B26:26/0  "REMOVE ME"
  B26:26/1  "REMOVE ME"
  B26:26/2  "REMOVE ME"
  B26:26/3  "REMOVE ME"
  B26:26/5  "REMOVE ME"
  B26:26/15  "REMOVE ME"
  B26:28/4  "REMOVE ME"
  B29:0/3  "REMOVE ME"
  B29:0/6  "REMOVE ME"
  B30:0  CONFIG_BITS_HARDWARE  "CONFIG Hardware options installed"
  B30:0/7  OUTLET_PX_INSTALLED  "PX-3 Installed"
  B30:0/10  CAB_SW_INSTALLED
  B30:1  CONF_BITS_HARDWARE_2
  B30:1/0  PS_24V_ENABLE
  B30:5  SYSTEM_STATUS_0  "STATUS System Status of system contro entities"
  B30:5/9  Z_PURGE_INIT
  B31:2  SYSTEM_HMI_CMD_0  "COMMAND HMI Commands"
  B31:3  SYSTEM_HMI_CMD_1  "COMMAND HMI Commands"
  B31:3/10  DEF_LP_INLET_GAS
  B31:4  SYSTEM_HMI_CMD_2  "COMMAND HMI Commands"
  B31:5  SYSTEM_HMI_CMD_3
  B31:6  SYSTEM_HMI_CMD_4  "COMMAND HMI Commands"
  B31:7  SYSTEM_HMI_CMD_5  "COMMAND HMI Commands"
  B31:8  SYSTEM_HMI_CMD_6  "COMMAND HMI Commands"
  B33:0  PURIFY_HMI_CMDS
  B33:0/1  DEF_PURIFY_MAX
  B34:0  REGEN_HMI_CMDS
  B34:1/1  HIGH_INLET_FLW
  B34:2  REGEN_FLAGS
  B34:3  REGEN_DEF_BUTTONS
  B35:2  MANUAL_HMI_CMNDS_0
  B36:0  PURGE_DEF_BUTTONS
  B36:1  PURGE_FLAGS
  B36:1/0  PURGE_VENT_ADS_DONE
  B36:1/1  PURGE_VENT_GET_DONE
  B36:1/3  PURGE_BACKFILL_DONE
  B36:1/4  PURGE_VENT_ADS_2_DN
  B36:1/5  PURGE_VENT_GET_2_DN
  B99:0/0  SIM_TEST_START
  B99:0/1  SIM_TEST_PURGE
  B99:0/2  SIM_B2  "Testing new code change. If correct delete this branch."
  B202:0  HMI_GETTER_STATUS
  C5:8  REGEN_PURGE_MINUTES  "COUNTER Regen THe number of minutes the purge step runs"
  DFILE:0  "OUTPUT"
  DFILE:1  "INPUT"
  DFILE:2  "STATUS"
  DFILE:3  "BINARY"
  DFILE:4  "TIMER"
  DFILE:5  "COUNTER"
  DFILE:6  "CONTROL"
  DFILE:7  "SYSTEM CFG Maintains the values that characterize t he system"
  DFILE:8  "FLOAT"
  DFILE:9  "CONSTANTS The collection of sy stem and subsystem c onstants"
  DFILE:10  "SYSTEM Contain the values f or system control"
  DFILE:11  "PROCESS Contains the values for the processing m achine"
  DFILE:12  "PURIFY Contains the values required for purify"
  DFILE:13  "REGEN Contains the values required for regen"
  DFILE:14  "BLIND N Blind Purge Integer File"
  DFILE:15  "MANUAL CTL Contains the data fo r the manual valve c ontrol"
  DFILE:16  "ADSORBER_A Contains the values for Adsorber A"
  DFILE:17  "ADSORBER_B Contains the values required for Adsorbe r B"
  DFILE:18  "GETTER CMN"
  DFILE:19  "BYPASS"
  DFILE:20  "PURGE"
  DFILE:21  "STARTUP"
  DFILE:22  "STARTUP"
  DFILE:23  "GETTER 1"
  DFILE:24  "PREHEATER"
  DFILE:25  "PID HTRS"
  DFILE:26  "FAULTS"
  DFILE:27  "QUICK STRT"
  DFILE:29  "GETTER"
  DFILE:30  "SYSTEM CFG"
  DFILE:31  "SYSTEM"
  DFILE:32  "PROCESS"
  DFILE:33  "PURIFY"
  DFILE:34  "REGEN"
  DFILE:35  "MANUAL CTL"
  DFILE:36  "PURGE"
  DFILE:37  "ADSORBER_B"
  DFILE:38  "BYPASS"
  DFILE:51  "LONG"
  DFILE:60  "READ_SBC"
  DFILE:61  "WRITE_SBC"
  DFILE:64  "MODBUS"
  DFILE:68  "COMMS"
  DFILE:69  "REVERSE"
  DFILE:99  "SIM_TEST"
  DFILE:200  "STATUS_SYS HMI System Status"
  DFILE:201  "STATUS_PUR HMI Status Purifier"
  DFILE:202  "STATUS_GET HMI STATUS Getter"
  DFILE:203  "STATUS_ADS HMI Status Adsorber"
  DFILE:206  "FLOAT_PRC HMI Purify function FLoat Values"
  DFILE:207  "STATUS_PRC HMI Purify Process f unction status"
  DFILE:210  "BUZZER Buzzer control"
  DFILE:250  "BLIND B Blind Purge Binary F ile"
  DFILE:251  "BLIND N Blind Purge Integer File"
  DFILE:252  "BLIND T Blind Purge Timer Fi le"
  DFILE:253  "BLIND C Blind Cycle Purge Co unter File"
  F8:1  TOTAL_FLOW_TEMP_CALC
  FIRST_SCAN  
  I:0.0/3  Z_PURGE_ALARM  "K2 - Normally closed. Inverse of K1 to provide a failsafe signal from Z-purge unit."
  I:0.0/4  PS1_STATUS
  I:0.0/5  PS2_STATUS
  I:0.0/9  X_PURGE_PRS_OK  "AUX 2 - Normally Closed. Signal high when pressure is above minimum required."
  I:0.0/11  Z_PURGE_OK_DEL
  I:1.0/0  ARGON_PRESS_SWITCH  "PS-1"
  I:1.0/5  WATER_FLOW_SWITCH  "FS-1"
  I:1.0/15  DIFF_PRESS_SWITCH
  N7:1  CONFIG_BITS_ALM_O  "CONFIG System alarms enable"
  N7:2  CONFIG_BITS_ALM_1  "CONFIG System alarms enable"
  N7:3  CONFIG_BITS_WARN_0  "CONFIG System warnings enable"
  N7:4  CONFIG_BITS_WARN_1  "CONFIG System warnings enable"
  N7:62  HP_GAS_ALM_HMI_SP  "High pressure alarm set in the HMI as an option"
  N7:63  HP_GAS_WARN_CALC_SP  "High pressure warninig calc thru "HP_GAS_ALM_SP""
  N7:70  LP_INLET_GAS_ALM_SP
  N7:71  LP_INLET_GAS_WRN_SP
  N7:98  LP_INT_PNEU_SP
  N10:6/14  LP_INLET_GAS_ALARM
  N10:8/14  LP_INLET_GAS_WARN
  N10:10  SYSTEM_CONTROL  "CONTROL System Bits used to manipulate hardware"
  N10:16  SYSTEM_FLAGS_1
  N10:16/6  MANUAL_CTRL_EXIT
  N10:19  INLET_PX_BAR
  N10:21  OUTLET_PX_BAR
  N10:31  ADS_A_INLET_PX_BAR
  N10:34  ADS_B_INLET_PX_BAR
  N10:37  PNEU_PX_BAR
  N10:41  ARGON_PX_BAR
  N10:44  PIPING_BAY_MB
  N11:2  PROC_ALARM_BUFFER  "STATE This holds the state of the process when the system alarm occured"
  N12:4  PURIFY_FLAGS_0  "STATUS Flags used by the purify process"
  N12:5  PURIFY_CONTROL  "CONTROL Control bits used by the purify process to change hardware states"
  N12:5/0  PURIFY_OPEN_IN_OUT  "CONTROL Purify Open the ADS purify in out valves"
  N12:6  PURIFY_COMPLETE  "STATUS Purify complete"
  N12:12  PURIFY_CALC_0  "CONFIG Math result placeholder for the purify time calculation"
  N12:13  PURIFY_FACTOR_TIME  "CONFIG The factored purify time accounting for the purify percent factor (hours)"
  N12:14  PURIFY_MAX_TIME
  N13:5  REGEN_CONTROL  "CONTROL Regen Bits used to manipulate hardware"
  N13:5/3  REGEN_OPEN_PROC_IN
  N13:5/8  REGEN_OPEN_EQUALIZE
  N13:6  REGEN_COMPLETE  "STATUS Regen complete"
  N13:8  BLANKET_LIMIT
  N13:12  ADS_PH_ROD_TC
  N14:0  QUICK_START_STATE
  N14:1  QUICK_STRT_STATE_BFR
  N15:4  MANUAL_FLAGS_0
  N16:3  ADS_A_FLAGS_0  "STATUS Flags used for Adsorber A"
  N16:17  PH_A_ROD_TEMP_READ
  N17:3  ADS_B_FLAGS_0  "STATUS Flags used for Adsorber B"
  N17:10  HMI_ADS_B_STATUS
  N17:16  HMI_ADS_B_STATUS2
  N17:17  PH_B_ROD_TEMP_READ
  N19:1  BYPASS_COMMAND  "HMI Commands received from the HMI"
  N21:51/0  QUICK_START_VENT
  N21:51/1  QUICK_START_BACKFILL
  N21:52  QUICK_REG_RUN_TIME
  N21:53  QUICK_REG_BLEED_FLW
  N21:54  QUICK_REG_BKFIL_FLW
  N23:9  GET_1_PH_SS_OUT_BUFF
  N24:5  "REMOVE ME"
  N24:6  "REMOVE ME"
  N24:10  "REMOVE ME"
  N24:11  "REMOVE ME"
  N24:12  "REMOVE ME"
  N24:13  "REMOVE ME"
  N24:14  "REMOVE ME"
  N203:0  "HMI Status word for Adsorber A"
  N203:1  "HMI Status word for Adsorber B"
  N220:0  HMI_STATUS_ADS_A1  "HMI Status Adsorber A Status Word"
  N220:1  P  "HMI Status Adsorber B Status Word"
  N220:4  STS_ADSA_OFFLINE
  N220:5  STS_ADSA_VENTING
  N220:6  STS_ADSA_BACKFILL
  N220:7  STS_ADSA_OFFLINE2
  N220:8  STS_ADSA_PUR_STANDBY
  N220:9  STS_ADSA_REG_OFFLINE
  N220:10  STS_ADSA_PUR_COOLING
  N220:11  STS_ADSA_PUR_VENTING
  N220:12  STS_ADSA_PUR_BACKFIL
  N220:13  STS_ADSA_PURIFYING
  N220:14  STS_ADSA_PUR_COOLIN2
  N220:15  STS_ADSA_PUR_VNTING2
  N220:16  STS_ADSA_PUR_VNTING3
  N220:17  STS_ADSA_REG_BACKFIL
  N220:18  STS_ADSA_REG_STANDBY
  N220:19  STS_ADSA_REG_PUR
  N220:20  STS_ADSA_PURIFYNG1
  N220:21  STS_ADSA_REG_VENTING
  N220:22  STS_ADSA_REG_HEATING
  N220:23  STS_ADSA_REG_HEATOFF
  N220:24  STS_ADSA_REGENERATIN
  N220:25  STS_ADSA_HEATERSOFF2
  N220:26  STS_ADSA_REG_COOLING
  N220:27  STS_ADSA_REG_BCKFIL2
  N220:28  STS_ADSA_REG_STNDBY2
  O:3.0/10  CUSTOM_IEC_EX_BYPASS  "Custom Bypass the IEC Ex X-Purge"
  PD25:6  "REMOVE ME"
  PD25:7  "REMOVE ME"
  T4:58  "REMOVE ME"
  T4:92  LP_INLET_GAS_ALM_TMR
  T4:93  LP_INLET_GAS_WRN_TMR
  T4:115  "REMOVE ME"
  T4:132  OPEN_TC11_ALM_TMR
  T4:137  OPEN_TC16_ALM_TMR
  T4:143  OPEN_TC16_WRN_TMR
  T4:148  OPEN_TC11_WRN_TMR
  T4:154  REGEN_STANDBY_DELAY
  T48:0  REGEN_EQUALIZE_SEC
  U:30  GETTER_2
  U:50  PLC_FAULT

COMMENTS NOT ATTACHED TO A CURRENT RUNG
  N7:8: Scale analog inputs / TODO: Do we need to add the ability to adjust the ammonia sensor scaling?
  N10:5/2: H2 SENSOR START UP DELAY / The H2 Sensor takes some time warm up until it can detect. The first scan triggers the H2 Sensor Start up delay until the H2 signal is on. The H2 sensor start up delay turns off at this time.
  RUNG000021-000020: End
  RUNG000023-000019: ADS B Wall Temp Thermocouple warning
  RUNG000023-000020: End
  T4:94: Startup Delay Timer
  B31:17/2: H2 SENSOR START UP DELAY / The H2 Sensor takes time to warm up. When the first scan is detected the system waits for the sensor value to come on before clearing the H2 Sensor start up delay warning.
  N7:109: DEFAULT PID SETTINGS
  T4:55: Preheater Fail to Heat
  PD25:0.0/3: Create output limit to maintain heating, but reduce rod limiting during startup. CVH = 50%, CVL = 35%, and OL is latched if PV<100 deg. C and unlatched if PV>180 deg. C
  N10:26: MFM / CONFIGURE MFM AND FLOW
  N203:0: BACKFILL = 7 (GREEN)
  B34:2/3: SBC in REGEN flag
  B3:0/2: Load BAR as default display value
  B34:3/0: Start REGEN on an EXOTHERMED bed after an EXOTHERM triggered bed swap.
  N7:3/4: If the alarm is not enabled for a specified amount of time, turn it back on.
  N10:25: MASS FLOW METER
  N220:0: BACKFILL = 7
  N20:0: Blind Purge Step 3: Vent Getter / Vent Getter based on a 10 minute timer instead of PX readings.

REVISION NOTES
  0: moved some bits out of N7 into B30
  1: moved bits out of N10 into B31
  2: moved bits from N15 into B35
  3: added the final data files. didn't need to move any bits
  4: updated configuration for TC and AI cards. updated DO module point assignments
  5: added logic for double-acting purify valves
  6: added rod and blanket limits
  7: added tags for default buttons
  8: cleaning up bed b pid control code
  9: removed h2 sensor and moved moisture sensor to channel 6
  10: changed processor name
  11: added px3 reading
  12: added call to mix panel routine
  13: test ok
  14: trying to clear plc fault by entering new pid default parameters
  15: changed stored PID values so that it maybe doesn't fault the PLC
  16: copid in new PID values from PS21
  17: cleared out the data table
  18: changed ADS_TC_OPEN_SP to 13700 by default
  19: setting default PID parameters
  20: added in preheater and blanket setpoints
  21: lots of changes to PID control
  22: fixed up PID defaults
  23: done testing
  24: got rid of separate PID defaults
  25: fixed loop update time bug in preheater defaults
  26: PID control done
  27: ok, now it's done. made Adsorber B use the same PID parameters as Adsorber A.
  28: added control for AV11 to system routine
  29: moved mixing panel valves into mixing panel routine
  30: some small fixes to the processing subroutine.
  31: cleaned up manual valve control for AV10, 11
  32: minor edit to purify factor calculation
  33: made some fixes to ADS_A routine including adding another state buffer for adsorber-only alarms.
  34: fixed up ADS_B routine so that it's like ADS_B
  35: Regen sequence modified and default regen paramters added
  36: added regen default comments
  37: added regen steps to constants
  38: Regen counter condition resets added
  39: Fixed regen standby buffer
  40: Regen buffering and sequencing checked and fixed
  41: Merged
  42: remove alarm aknowledge
  43: Updated alarm tag names
  44: PH fault changed
  45: manual mode PID taop PID control
  46: Added fail to cool alarm and warning
  47: trying to fix ph fault
  48: fixing open tc
  49: fixed open tc logic
  50: ok, now it's fixed

DATA TABLE (non-zero values as saved)
DATA T4
% .PRE .ACC %
% T4:0 % 2 0
% T4:1 % 60 0
% T4:2 % 2 0
% T4:3 % 10 0
% T4:4 % 60 0
% T4:5 % 60 0
% T4:6 % 1000 0
% T4:7 % 1000 0
% T4:8 % 5 0
% T4:9 % 5 0
% T4:10 % 5 0
% T4:11 % 5 0
% T4:12 % 5 0
% T4:13 % 60 0
% T4:14 % 5 0
% T4:15 % 60 0
% T4:16 % 18000 0
% T4:17 % 18000 0
% T4:18 % 18000 0
% T4:19 % 18000 0
% T4:20 % 5 0
% T4:21 % 60 0
% T4:22 % 5 0
% T4:23 % 60 0
% T4:24 % 1 0
% T4:25 % 1 0
% T4:26 % 5 0
% T4:27 % 5 0
% T4:28 % 5 0
% T4:29 % 5 0
% T4:30 % 60 0
% T4:31 % 60 0
% T4:32 % 5 0
% T4:33 % 5 0
% T4:34 % 2 0
% T4:35 % 5 0
% T4:36 % 5 0
% T4:37 % 5 0
% T4:38 % 5 0
% T4:39 % 5 0
% T4:40 % 5 0
% T4:41 % 5 0
% T4:42 % 5 0
% T4:43 % 5 0
% T4:44 % 60 0
% T4:45 % 120 0
% T4:46 % 60 0
% T4:47 % 120 0
% T4:48 % 60 0
% T4:49 % 60 0
% T4:50 % 60 0
% T4:51 % 60 60
% T4:52 % 2 0
% T4:53 % 2 0
% T4:54 % 60 0
% T4:55 % 60 0
% T4:56 % 2 0
% T4:57 % 2 0
% T4:58 % 2 0
% T4:59 % 100 0
% T4:60 % 5 0
% T4:61 % 5 0
% T4:62 % 5 0
% T4:63 % 5 0
% T4:64 % 5 0
% T4:65 % 5 0
% T4:66 % 5 0
% T4:67 % 5 0
% T4:68 % 5 0
% T4:69 % 5 0
% T4:70 % 5 0
% T4:71 % 5 0
% T4:72 % 5 0
% T4:73 % 5 0
% T4:74 % 60 0
% T4:75 % 60 0
% T4:76 % 60 0
% T4:77 % 60 0
% T4:78 % 5 0
% T4:79 % 5 0
% T4:80 % 5 0
% T4:81 % 5 0
% T4:82 % 5 0
% T4:84 % 5 0
% T4:86 % 5 0
% T4:88 % 5 0
% T4:90 % 500 0
% T4:91 % 5 0
% T4:92 % 5 0
% T4:93 % 5 0
% T4:94 % 2 0
% T4:95 % 2 0
% T4:96 % 5 0
% T4:97 % 5 0
% T4:98 % 5 0
% T4:99 % 5 0
% T4:100 % 5 0
% T4:101 % 180 180
% T4:102 % 2 2
% T4:103 % 240 0
% T4:104 % 60 0
% T4:105 % 60 0
% T4:106 % 30 0
% T4:107 % 60 0
% T4:108 % 5 0
% T4:109 % 60 0
% T4:110 % 5 0
% T4:111 % 60 0
% T4:112 % 5 0
% T4:113 % 5 0
% T4:114 % 300 0
% T4:115 % 300 0
% T4:116 % 1000 0
% T4:117 % 1000 0
% T4:119 % 5 0
% T4:121 % 5 0
% T4:122 % 5 0
% T4:123 % 5 0
% T4:124 % 5 0
% T4:125 % 5 0
% T4:126 % 5 0
% T4:127 % 5 0
% T4:128 % 5 0
% T4:129 % 5 0
% T4:130 % 5 0
% T4:131 % 5 0
% T4:133 % 5 0
% T4:134 % 5 0
% T4:135 % 5 0
% T4:136 % 5 0
% T4:138 % 30 0
% T4:139 % 5 0
% T4:140 % 5 0
% T4:141 % 5 0
% T4:142 % 5 0
% T4:144 % 5 0
% T4:145 % 5 0
% T4:146 % 5 0
% T4:147 % 5 0
% T4:149 % 30 0
% T4:150 % 1000 0
% T4:151 % 1000 33
% T4:152 % 100 44
% T4:153 % 100 0
% T4:154 % 1 0
% T4:155 % 2 2
% T4:156 % 60 21
% T4:157 % 5 0
% T4:158 % 5 0
% T4:159 % 5 0
% T4:160 % 5 0
% T4:161 % 500 0
% T4:162 % 500 0
% T4:164 % 5 0
% T4:165 % 5 0
% T4:166 % 5 0
% T4:167 % 60 0
DATA C5
% .PRE .ACC %
% C5:0 % 48 0
% C5:1 % 60 0
% C5:2 % 24 21
% C5:3 % 32767 0
% C5:4 % 480 0
% C5:5 % 120 0
% C5:7 % 12 0
% C5:8 % 480 0
% C5:9 % 30 0
% C5:10 % 30 0
% C5:11 % 30 0
% C5:12 % 300 0
% C5:13 % 300 0
% C5:14 % 12 0
% C5:15 % 10 0
% C5:16 % 32767 0
% C5:17 % 480 0
% C5:18 % 480 0
% C5:19 % 27 4
% C5:20 % 16 16
% C5:21 % 30 0
% C5:22 % 30 0
DATA R6
% .LEN .POS %
% R6:0 % 16 0
% R6:1 % 16 0
DATA N64
% N64:0 % -24188 0 0 0 0 0 0 0 0 0
DATA T252
% .PRE .ACC %
% T252:0 % 60 0
% T252:1 % 60 0
% T252:2 % 60 0
% T252:3 % 60 0
% T252:4 % 60 0
DATA C253
% .PRE .ACC %
% C253:0 % 10 0
% C253:1 % 10 0
% C253:2 % 10 0
% C253:3 % 10 0
% C253:4 % 10 0
% C253:5 % 10 0
